// TIA Portal V18 export
FUNCTION_BLOCK "FB10-Condition Check_1"   // FB14, LAD
{ S7_Optimized_Access := 'TRUE' }
VERSION : 0.1
// stored: AutoNumber true, IsIECCheckEnabled false, IsRetainMemResEnabled false, MemoryReserve 100, SetENOAutomatically false, UDAEnableTagReadback false
   VAR_INPUT
      "Time" : DInt;
      "Pump ON delay" : DInt;
      Check_Time { ExternalAccessible := 'False'; ExternalVisible := 'False'; ExternalWritable := 'False'} : DInt;
      Pressure_SP { ExternalAccessible := 'False'; ExternalVisible := 'False'; ExternalWritable := 'False'} : Real;
      Pressure_tolerance { ExternalAccessible := 'False'; ExternalVisible := 'False'; ExternalWritable := 'False'} : Real;
      Current_pressure { ExternalAccessible := 'False'; ExternalVisible := 'False'; ExternalWritable := 'False'} : Real;
      selected { ExternalAccessible := 'False'; ExternalVisible := 'False'; ExternalWritable := 'False'} : Bool;
      "Pressurising Tolerance" : Real;
      Pressurising_SP : Real;
   END_VAR
   VAR_OUTPUT
      "dispensing Time PV" : Int;
      "Checking Time pv" { ExternalAccessible := 'False'; ExternalVisible := 'False'; ExternalWritable := 'False'} : Int;
      Leaktest_ok { ExternalAccessible := 'False'; ExternalVisible := 'False'; ExternalWritable := 'False'} : Bool;
      Leaktest_nok { ExternalAccessible := 'False'; ExternalVisible := 'False'; ExternalWritable := 'False'} : Bool;
      Conditiontest_OK : Bool;
      Conditiontest_NOK { ExternalAccessible := 'False'; ExternalVisible := 'False'; ExternalWritable := 'False'} : Bool;
      "PAT @ installation" : DInt;   // Pressure achieved Time @ Installation
      Test_Data : "Condition_Check";
   END_VAR
   VAR_IN_OUT
      Commissioning_mode : Bool;
      "Start ConditonCheck" : Bool;
      "Stop ConditonCheck" : Bool;
      "ConditonCheck Running" : Bool;
      "ConditonCheck completed" : Bool;
      "ON Gear Pump" : Bool;
      "ON inlet" : Bool;
      Pressurising : Bool;
      run_rev : Bool;
   END_VAR
   VAR
      "dispensing time done" : Bool;
      "dispensing time in sec" : DInt;
      "timer input" : DInt;
      IEC_Timer_0_Instance_1 { S7_SetPoint := 'True'} : TON_TIME;
      IEC_Timer_0_Instance_2 { S7_SetPoint := 'True'} : TON_TIME;
      IEC_Timer_0_Instance_4 { S7_SetPoint := 'True'} : TON_TIME;
      "Press+ve" { ExternalAccessible := 'False'; ExternalVisible := 'False'; ExternalWritable := 'False'; S7_SetPoint := 'True'} : Real;
      "Press-ve" { ExternalAccessible := 'False'; ExternalVisible := 'False'; ExternalWritable := 'False'} : Real;
      IEC_Timer_0_Instance_3 { ExternalAccessible := 'False'; ExternalVisible := 'False'; ExternalWritable := 'False'; S7_SetPoint := 'True'} : TON_TIME;
      Checktime_ms { ExternalAccessible := 'False'; ExternalVisible := 'False'; ExternalWritable := 'False'; S7_SetPoint := 'True'} : DInt;
      Check_timesec { ExternalAccessible := 'False'; ExternalVisible := 'False'; ExternalWritable := 'False'} : DInt;
      temp_ons { ExternalAccessible := 'False'; ExternalVisible := 'False'; ExternalWritable := 'False'} : Bool;
      temp : Array[0..5] of Bool;
      IEC_Timer_0_Instance_5 { S7_SetPoint := 'True'} : TON_TIME;
      "WIth Tolerance" { S7_SetPoint := 'True'} : DInt;
      Pressure_achive_time : DInt;
      Pressure_ok : Bool;
      IEC_Timer_0_Instance { S7_SetPoint := 'True'} : TON_TIME;
      Result { S7_SetPoint := 'True'} : Bool;
      "result temp" : Bool;
      IEC_Timer_0_Instance_6 { S7_SetPoint := 'True'} : TON_TIME;
      Start_cond : Bool;
      IEC_Timer_0_Instance_7 { S7_SetPoint := 'True'} : TON_TIME;
   END_VAR
   VAR_TEMP
      ret : Int;
   END_VAR
   VAR_TEMP   // added for the SCL form of the ladder/FBD networks
      _w1 : Bool;
      _w2 : Bool;
      _w3 : Bool;
      _w4 : Bool;
      _w5 : Bool;
   END_VAR
BEGIN

REGION Network 1
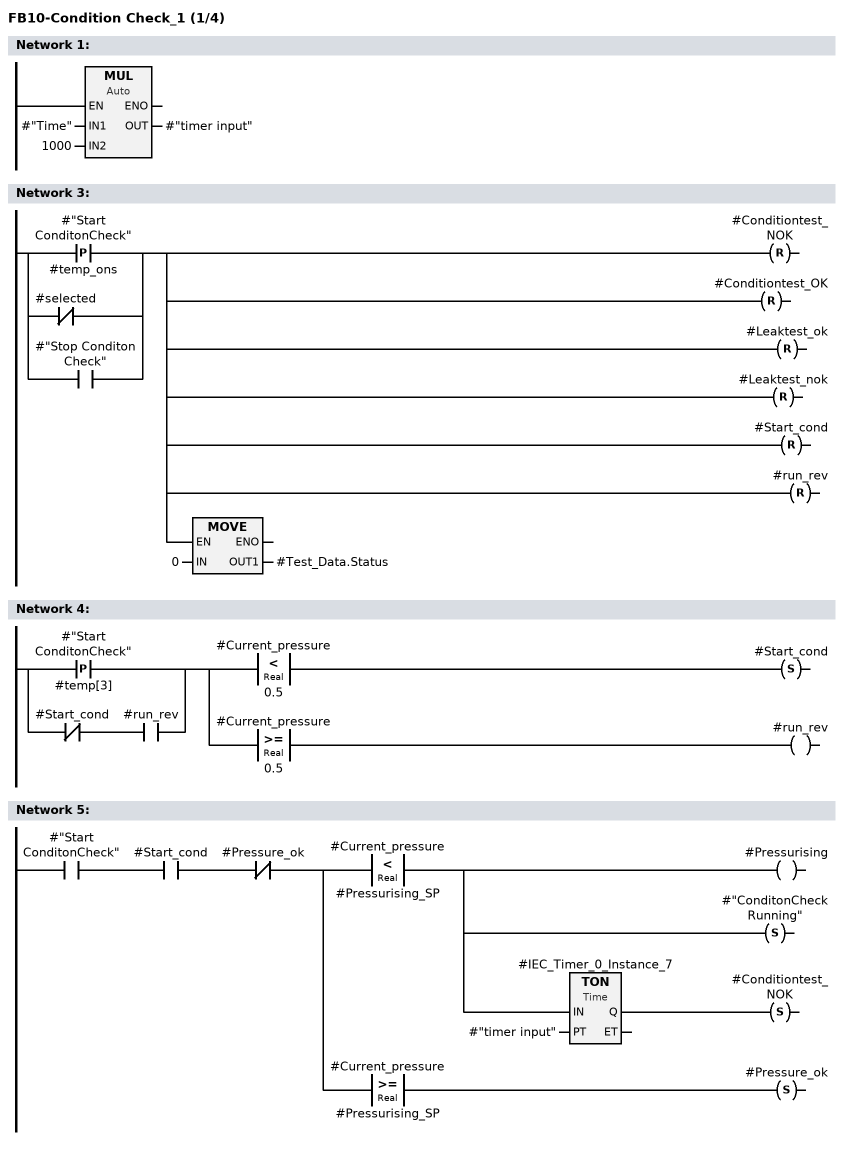
   RUNG wire#powerrail
      Mul(in1 := #"Time", in2 := 1000, out => #"timer input")
   END_RUNG
   // the same network as SCL:
   #"timer input" := #"Time" * 1000;
END_REGION

REGION Network 2 (SCL)
   #"WIth Tolerance" := ROUND(#"PAT @ installation" + ((#"PAT @ installation"*#"Pressurising Tolerance")/100));
END_REGION

REGION Network 3
   RUNG wire#powerrail
      P_Contact(operand := #"Start ConditonCheck", bit := #temp_ons)
      wire#w1
      R_Coil( #Conditiontest_NOK )
   END_RUNG
   RUNG wire#powerrail
      I_Contact( #selected )
   END_RUNG wire#w1
   RUNG wire#powerrail
      Contact( #"Stop ConditonCheck" )
   END_RUNG wire#w1
   RUNG wire#w1
      R_Coil( #Conditiontest_OK )
   END_RUNG
   RUNG wire#w1
      R_Coil( #Leaktest_ok )
   END_RUNG
   RUNG wire#w1
      R_Coil( #Leaktest_nok )
   END_RUNG
   RUNG wire#w1
      R_Coil( #Start_cond )
   END_RUNG
   RUNG wire#w1
      R_Coil( #run_rev )
   END_RUNG
   RUNG wire#w1
      Move(in := 0, out1 => #Test_Data.Status)
   END_RUNG
   // the same network as SCL:
   #_w1 := #"Start ConditonCheck" AND NOT #temp_ons;   // rising edge of #"Start ConditonCheck"
   #temp_ons := #"Start ConditonCheck";
   IF #_w1 OR NOT #selected OR #"Stop ConditonCheck" THEN
       #Conditiontest_NOK := FALSE;
       #Conditiontest_OK := FALSE;
       #Leaktest_ok := FALSE;
       #Leaktest_nok := FALSE;
       #Start_cond := FALSE;
       #run_rev := FALSE;
       #Test_Data.Status := 0;
   END_IF;
END_REGION

REGION Network 4
   RUNG wire#powerrail
      P_Contact(operand := #"Start ConditonCheck", bit := #temp[3])
      wire#w1
      { S7_Templates := "SrcType := Real" } LT_Contact(in1 := #Current_pressure, in2 := 0.5)
      S_Coil( #Start_cond )
   END_RUNG
   RUNG wire#powerrail
      I_Contact( #Start_cond )
      Contact( #run_rev )
   END_RUNG wire#w1
   RUNG wire#w1
      { S7_Templates := "SrcType := Real" } GE_Contact(in1 := #Current_pressure, in2 := 0.5)
      Coil( #run_rev )
   END_RUNG
   // the same network as SCL:
   #_w1 := #"Start ConditonCheck" AND NOT #temp[3];   // rising edge of #"Start ConditonCheck"
   #temp[3] := #"Start ConditonCheck";
   #_w2 := #_w1 OR (NOT #Start_cond AND #run_rev);
   IF #_w2 AND (#Current_pressure < 0.5) THEN #Start_cond := TRUE; END_IF;
   #run_rev := #_w2 AND (#Current_pressure >= 0.5);
END_REGION

REGION Network 5
   RUNG wire#powerrail
      Contact( #"Start ConditonCheck" )
      Contact( #Start_cond )
      I_Contact( #Pressure_ok )
      wire#w1
      { S7_Templates := "SrcType := Real" } LT_Contact(in1 := #Current_pressure, in2 := #Pressurising_SP)
      wire#w2
      Coil( #Pressurising )
   END_RUNG
   RUNG wire#w2
      S_Coil( #"ConditonCheck Running" )
   END_RUNG
   RUNG wire#w2
      { S7_Templates := "time_type := Time" } #IEC_Timer_0_Instance_7.TON(pt := #"timer input", et =>)
      S_Coil( #Conditiontest_NOK )
   END_RUNG
   RUNG wire#w1
      { S7_Templates := "SrcType := Real" } GE_Contact(in1 := #Current_pressure, in2 := #Pressurising_SP)
      S_Coil( #Pressure_ok )
   END_RUNG
   // the same network as SCL:
   #_w1 := #"Start ConditonCheck" AND #Start_cond AND NOT #Pressure_ok;
   #Pressurising := #_w1 AND (#Current_pressure < #Pressurising_SP);
   IF #Pressurising THEN #"ConditonCheck Running" := TRUE; END_IF;
   #IEC_Timer_0_Instance_7(IN := #Pressurising, PT := #"timer input");   // TON
   IF #IEC_Timer_0_Instance_7.Q THEN #Conditiontest_NOK := TRUE; END_IF;
   IF #_w1 AND (#Current_pressure >= #Pressurising_SP) THEN #Pressure_ok := TRUE; END_IF;
END_REGION

REGION Network 6
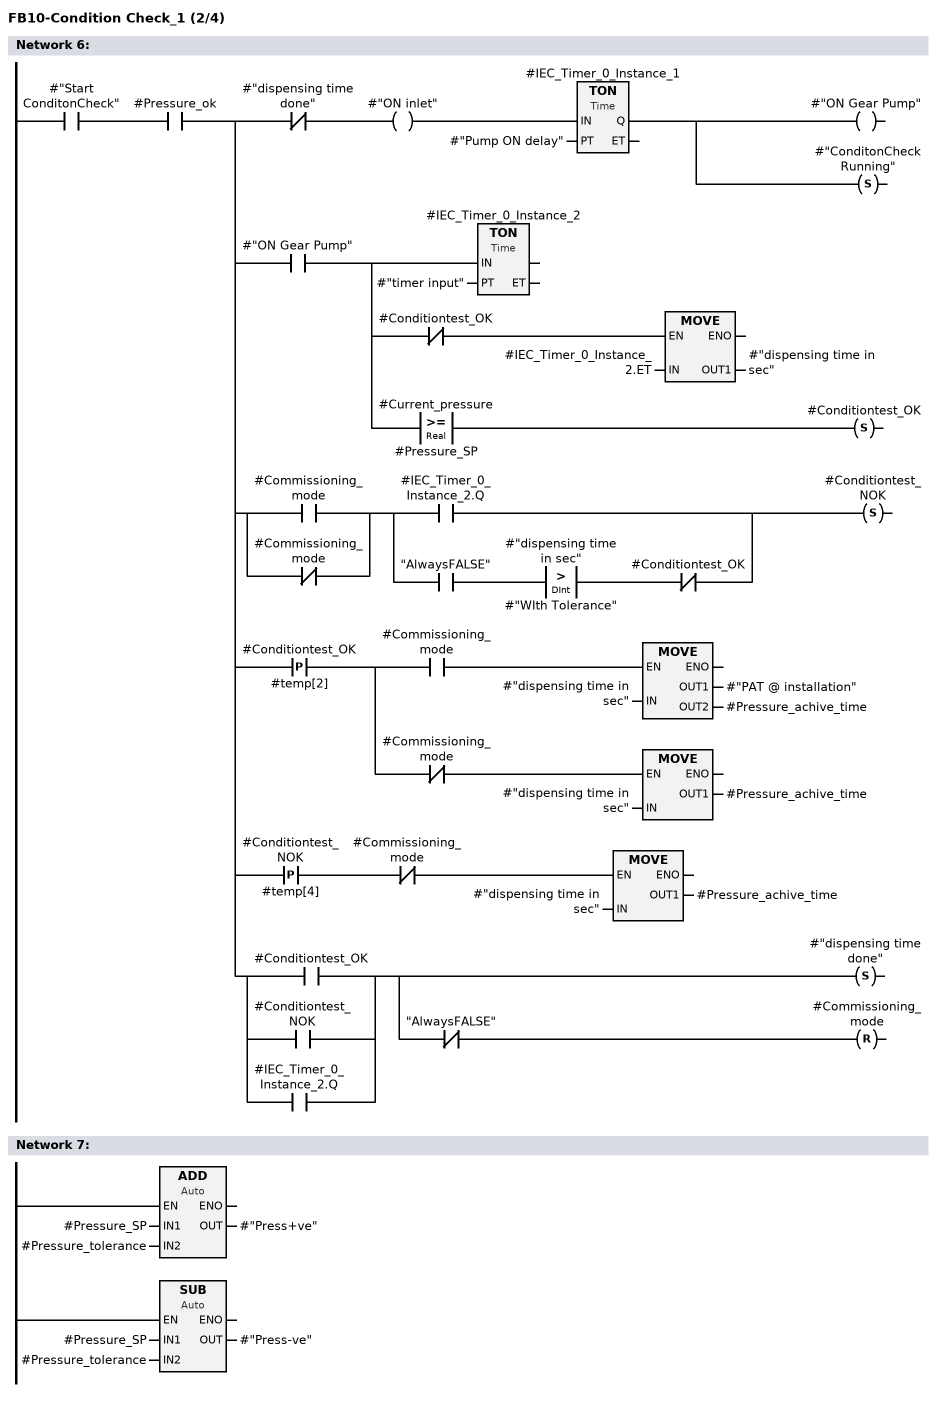
   RUNG wire#powerrail
      Contact( #"Start ConditonCheck" )
      Contact( #Pressure_ok )
      wire#w1
      I_Contact( #"dispensing time done" )
      Coil( #"ON inlet" )
      { S7_Templates := "time_type := Time" } #IEC_Timer_0_Instance_1.TON(pt := #"Pump ON delay", et =>)
      wire#w2
      Coil( #"ON Gear Pump" )
   END_RUNG
   RUNG wire#w2
      S_Coil( #"ConditonCheck Running" )
   END_RUNG
   RUNG wire#w1
      Contact( #"ON Gear Pump" )
      wire#w3
      { S7_Templates := "time_type := Time" } #IEC_Timer_0_Instance_2.TON(pt := #"timer input", et =>)
   END_RUNG
   RUNG wire#w3
      I_Contact( #Conditiontest_OK )
      Move(in := #IEC_Timer_0_Instance_2.ET, out1 => #"dispensing time in sec")
   END_RUNG
   RUNG wire#w3
      { S7_Templates := "SrcType := Real" } GE_Contact(in1 := #Current_pressure, in2 := #Pressure_SP)
      S_Coil( #Conditiontest_OK )
   END_RUNG
   RUNG wire#w1
      Contact( #Commissioning_mode )
      wire#w4
      Contact( #IEC_Timer_0_Instance_2.Q )
      wire#w5
      S_Coil( #Conditiontest_NOK )
   END_RUNG
   RUNG wire#w1
      I_Contact( #Commissioning_mode )
   END_RUNG wire#w4
   RUNG wire#w4
      Contact( "AlwaysFALSE" )
      { S7_Templates := "SrcType := DInt" } GT_Contact(in1 := #"dispensing time in sec", in2 := #"WIth Tolerance")
      I_Contact( #Conditiontest_OK )
   END_RUNG wire#w5
   RUNG wire#w1
      P_Contact(operand := #Conditiontest_OK, bit := #temp[2])
      wire#w6
      Contact( #Commissioning_mode )
      Move(in := #"dispensing time in sec", out1 => #"PAT @ installation", out2 => #Pressure_achive_time)
   END_RUNG
   RUNG wire#w6
      I_Contact( #Commissioning_mode )
      Move(in := #"dispensing time in sec", out1 => #Pressure_achive_time)
   END_RUNG
   RUNG wire#w1
      P_Contact(operand := #Conditiontest_NOK, bit := #temp[4])
      I_Contact( #Commissioning_mode )
      Move(in := #"dispensing time in sec", out1 => #Pressure_achive_time)
   END_RUNG
   RUNG wire#w1
      Contact( #Conditiontest_OK )
      wire#w7
      S_Coil( #"dispensing time done" )
   END_RUNG
   RUNG wire#w1
      Contact( #Conditiontest_NOK )
   END_RUNG wire#w7
   RUNG wire#w1
      Contact( #IEC_Timer_0_Instance_2.Q )
   END_RUNG wire#w7
   RUNG wire#w7
      I_Contact( "AlwaysFALSE" )
      R_Coil( #Commissioning_mode )
   END_RUNG
   // the same network as SCL:
   #_w1 := #"Start ConditonCheck" AND #Pressure_ok;
   #"ON inlet" := #_w1 AND NOT #"dispensing time done";
   #IEC_Timer_0_Instance_1(IN := #"ON inlet", PT := #"Pump ON delay");   // TON
   #"ON Gear Pump" := #IEC_Timer_0_Instance_1.Q;
   IF #IEC_Timer_0_Instance_1.Q THEN #"ConditonCheck Running" := TRUE; END_IF;
   #_w2 := #_w1 AND #"ON Gear Pump";
   #IEC_Timer_0_Instance_2(IN := #_w2, PT := #"timer input");   // TON
   IF #_w2 AND NOT #Conditiontest_OK THEN #"dispensing time in sec" := #IEC_Timer_0_Instance_2.ET; END_IF;
   IF #_w2 AND (#Current_pressure >= #Pressure_SP) THEN #Conditiontest_OK := TRUE; END_IF;
   IF #_w1 AND (#Commissioning_mode OR NOT #Commissioning_mode) AND (#IEC_Timer_0_Instance_2.Q OR ("AlwaysFALSE" AND (#"dispensing time in sec" > #"WIth Tolerance") AND NOT #Conditiontest_OK)) THEN
       #Conditiontest_NOK := TRUE;
   END_IF;
   #_w3 := #_w1 AND #Conditiontest_OK AND NOT #temp[2];   // rising edge of #Conditiontest_OK
   #temp[2] := #Conditiontest_OK;
   IF #_w3 AND #Commissioning_mode THEN
       #"PAT @ installation" := #"dispensing time in sec";
       #Pressure_achive_time := #"dispensing time in sec";
   END_IF;
   IF #_w3 AND NOT #Commissioning_mode THEN #Pressure_achive_time := #"dispensing time in sec"; END_IF;
   #_w4 := #_w1 AND #Conditiontest_NOK AND NOT #temp[4];   // rising edge of #Conditiontest_NOK
   #temp[4] := #Conditiontest_NOK;
   IF #_w4 AND NOT #Commissioning_mode THEN #Pressure_achive_time := #"dispensing time in sec"; END_IF;
   #_w5 := #_w1 AND (#Conditiontest_OK OR #Conditiontest_NOK OR #IEC_Timer_0_Instance_2.Q);
   IF #_w5 THEN #"dispensing time done" := TRUE; END_IF;
   IF #_w5 AND NOT "AlwaysFALSE" THEN #Commissioning_mode := FALSE; END_IF;
END_REGION

REGION Network 7
   RUNG wire#powerrail
      Add(in1 := #Pressure_SP, in2 := #Pressure_tolerance, out => #"Press+ve")
   END_RUNG
   RUNG wire#powerrail
      Sub(in1 := #Pressure_SP, in2 := #Pressure_tolerance, out => #"Press-ve")
   END_RUNG
   // the same network as SCL:
   #"Press+ve" := #Pressure_SP + #Pressure_tolerance;
   #"Press-ve" := #Pressure_SP - #Pressure_tolerance;
END_REGION

REGION Network 8
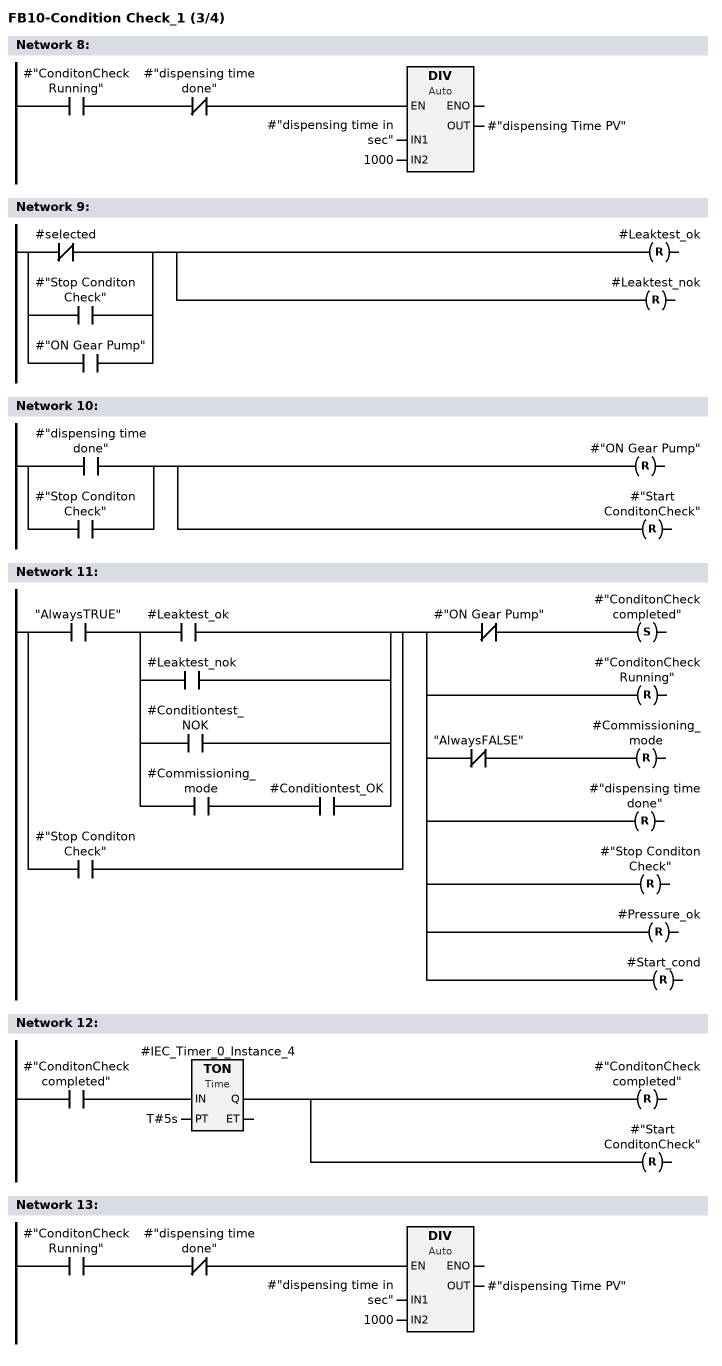
   RUNG wire#powerrail
      Contact( #"ConditonCheck Running" )
      I_Contact( #"dispensing time done" )
      Div(in1 := #"dispensing time in sec", in2 := 1000, out => #"dispensing Time PV")
   END_RUNG
   // the same network as SCL:
   IF #"ConditonCheck Running" AND NOT #"dispensing time done" THEN
       #"dispensing Time PV" := #"dispensing time in sec" / 1000;
   END_IF;
END_REGION

REGION Network 9
   RUNG wire#powerrail
      I_Contact( #selected )
      wire#w1
      R_Coil( #Leaktest_ok )
   END_RUNG
   RUNG wire#powerrail
      Contact( #"Stop ConditonCheck" )
   END_RUNG wire#w1
   RUNG wire#powerrail
      Contact( #"ON Gear Pump" )
   END_RUNG wire#w1
   RUNG wire#w1
      R_Coil( #Leaktest_nok )
   END_RUNG
   // the same network as SCL:
   IF NOT #selected OR #"Stop ConditonCheck" OR #"ON Gear Pump" THEN
       #Leaktest_ok := FALSE;
       #Leaktest_nok := FALSE;
   END_IF;
END_REGION

REGION Network 10
   RUNG wire#powerrail
      Contact( #"dispensing time done" )
      wire#w1
      R_Coil( #"ON Gear Pump" )
   END_RUNG
   RUNG wire#powerrail
      Contact( #"Stop ConditonCheck" )
   END_RUNG wire#w1
   RUNG wire#w1
      R_Coil( #"Start ConditonCheck" )
   END_RUNG
   // the same network as SCL:
   IF #"dispensing time done" OR #"Stop ConditonCheck" THEN
       #"ON Gear Pump" := FALSE;
       #"Start ConditonCheck" := FALSE;
   END_IF;
END_REGION

REGION Network 11
   RUNG wire#powerrail
      Contact( "AlwaysTRUE" )
      wire#w1
      Contact( #Leaktest_ok )
      wire#w2
      I_Contact( #"ON Gear Pump" )
      S_Coil( #"ConditonCheck completed" )
   END_RUNG
   RUNG wire#w1
      Contact( #Leaktest_nok )
   END_RUNG wire#w2
   RUNG wire#w1
      Contact( #Conditiontest_NOK )
   END_RUNG wire#w2
   RUNG wire#w1
      Contact( #Commissioning_mode )
      Contact( #Conditiontest_OK )
   END_RUNG wire#w2
   RUNG wire#powerrail
      Contact( #"Stop ConditonCheck" )
   END_RUNG wire#w2
   RUNG wire#w2
      R_Coil( #"ConditonCheck Running" )
   END_RUNG
   RUNG wire#w2
      I_Contact( "AlwaysFALSE" )
      R_Coil( #Commissioning_mode )
   END_RUNG
   RUNG wire#w2
      R_Coil( #"dispensing time done" )
   END_RUNG
   RUNG wire#w2
      R_Coil( #"Stop ConditonCheck" )
   END_RUNG
   RUNG wire#w2
      R_Coil( #Pressure_ok )
   END_RUNG
   RUNG wire#w2
      R_Coil( #Start_cond )
   END_RUNG
   // the same network as SCL:
   #_w1 := ("AlwaysTRUE" AND (#Leaktest_ok OR #Leaktest_nok OR #Conditiontest_NOK OR (#Commissioning_mode AND #Conditiontest_OK))) OR #"Stop ConditonCheck";
   IF #_w1 AND NOT #"ON Gear Pump" THEN #"ConditonCheck completed" := TRUE; END_IF;
   IF #_w1 THEN #"ConditonCheck Running" := FALSE; END_IF;
   IF #_w1 AND NOT "AlwaysFALSE" THEN #Commissioning_mode := FALSE; END_IF;
   IF #_w1 THEN
       #"dispensing time done" := FALSE;
       #"Stop ConditonCheck" := FALSE;
       #Pressure_ok := FALSE;
       #Start_cond := FALSE;
   END_IF;
END_REGION

REGION Network 12
   RUNG wire#powerrail
      Contact( #"ConditonCheck completed" )
      { S7_Templates := "time_type := Time" } #IEC_Timer_0_Instance_4.TON(pt := T#5s, et =>)
      wire#w1
      R_Coil( #"ConditonCheck completed" )
   END_RUNG
   RUNG wire#w1
      R_Coil( #"Start ConditonCheck" )
   END_RUNG
   // the same network as SCL:
   #IEC_Timer_0_Instance_4(IN := #"ConditonCheck completed", PT := T#5s);   // TON
   IF #IEC_Timer_0_Instance_4.Q THEN
       #"ConditonCheck completed" := FALSE;
       #"Start ConditonCheck" := FALSE;
   END_IF;
END_REGION

REGION Network 13
   RUNG wire#powerrail
      Contact( #"ConditonCheck Running" )
      I_Contact( #"dispensing time done" )
      Div(in1 := #"dispensing time in sec", in2 := 1000, out => #"dispensing Time PV")
   END_RUNG
   // the same network as SCL:
   IF #"ConditonCheck Running" AND NOT #"dispensing time done" THEN
       #"dispensing Time PV" := #"dispensing time in sec" / 1000;
   END_IF;
END_REGION

REGION Network 14
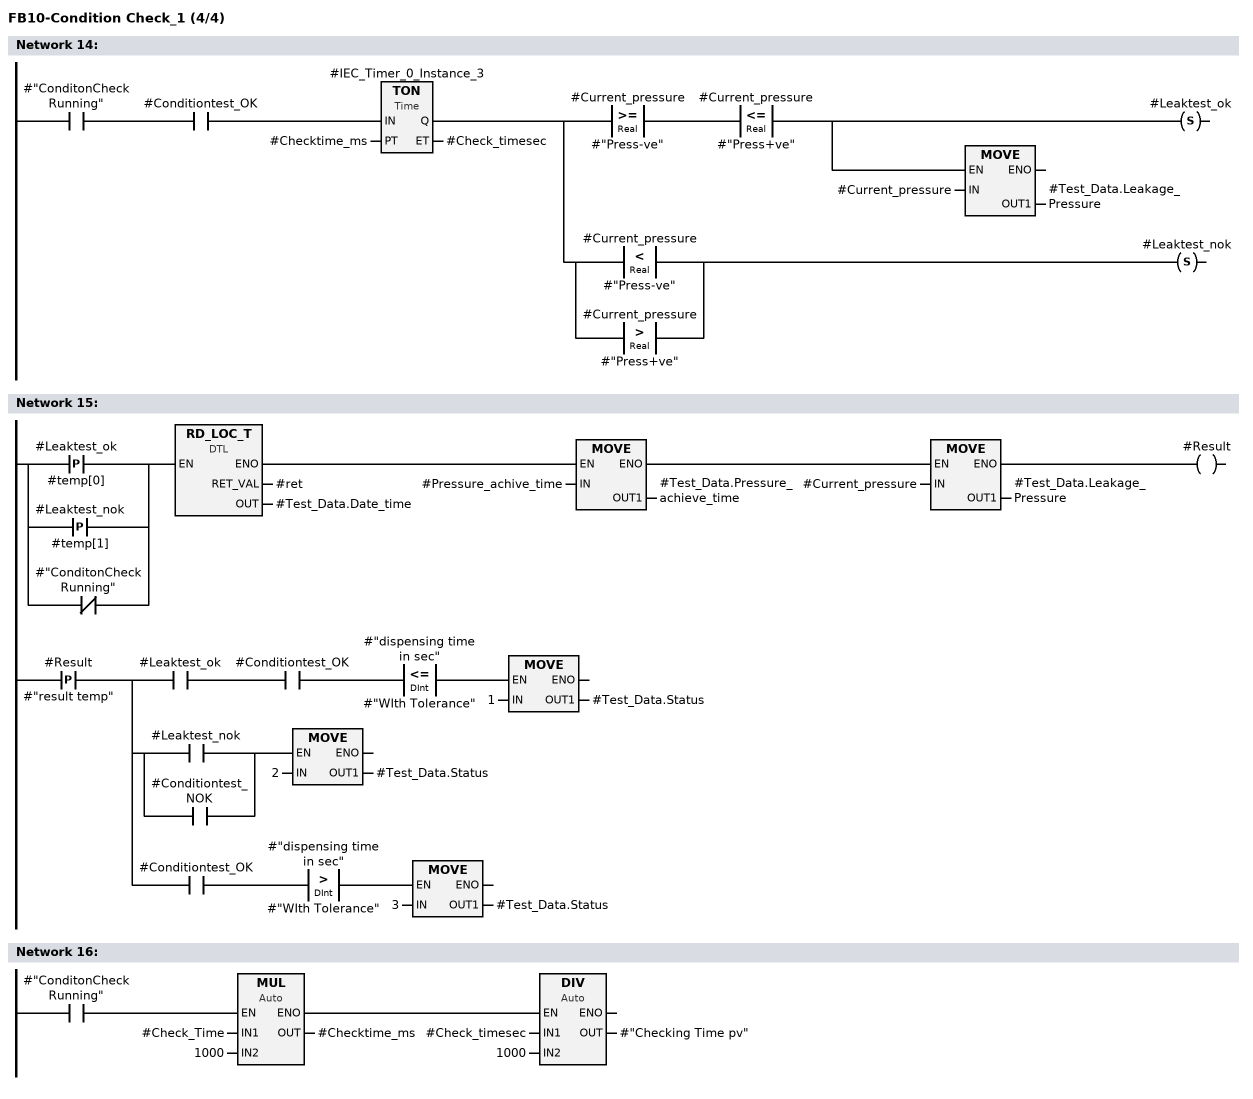
   RUNG wire#powerrail
      Contact( #"ConditonCheck Running" )
      Contact( #Conditiontest_OK )
      { S7_Templates := "time_type := Time" } #IEC_Timer_0_Instance_3.TON(pt := #Checktime_ms, et => #Check_timesec)
      wire#w1
      { S7_Templates := "SrcType := Real" } GE_Contact(in1 := #Current_pressure, in2 := #"Press-ve")
      { S7_Templates := "SrcType := Real" } LE_Contact(in1 := #Current_pressure, in2 := #"Press+ve")
      wire#w2
      S_Coil( #Leaktest_ok )
   END_RUNG
   RUNG wire#w2
      Move(in := #Current_pressure, out1 => #Test_Data.Leakage_Pressure)
   END_RUNG
   RUNG wire#w1
      { S7_Templates := "SrcType := Real" } LT_Contact(in1 := #Current_pressure, in2 := #"Press-ve")
      wire#w3
      S_Coil( #Leaktest_nok )
   END_RUNG
   RUNG wire#w1
      { S7_Templates := "SrcType := Real" } GT_Contact(in1 := #Current_pressure, in2 := #"Press+ve")
   END_RUNG wire#w3
   // the same network as SCL:
   #IEC_Timer_0_Instance_3(IN := #"ConditonCheck Running" AND #Conditiontest_OK,   // TON
                           PT := #Checktime_ms,
                           ET => #Check_timesec);
   IF #IEC_Timer_0_Instance_3.Q AND (#Current_pressure >= #"Press-ve") AND (#Current_pressure <= #"Press+ve") THEN
       #Leaktest_ok := TRUE;
       #Test_Data.Leakage_Pressure := #Current_pressure;
   END_IF;
   IF #IEC_Timer_0_Instance_3.Q AND ((#Current_pressure < #"Press-ve") OR (#Current_pressure > #"Press+ve")) THEN
       #Leaktest_nok := TRUE;
   END_IF;
END_REGION

REGION Network 15
   RUNG wire#powerrail
      P_Contact(operand := #Leaktest_ok, bit := #temp[0])
      wire#w1
      { S7_Templates := "date_type := DTL" } RD_LOC_T(RET_VAL => #ret, OUT => #Test_Data.Date_time)
      Move(in := #Pressure_achive_time, out1 => #Test_Data.Pressure_achieve_time)
      Move(in := #Current_pressure, out1 => #Test_Data.Leakage_Pressure)
      Coil( #Result )
   END_RUNG
   RUNG wire#powerrail
      P_Contact(operand := #Leaktest_nok, bit := #temp[1])
   END_RUNG wire#w1
   RUNG wire#powerrail
      I_Contact( #"ConditonCheck Running" )
   END_RUNG wire#w1
   RUNG wire#powerrail
      P_Contact(operand := #Result, bit := #"result temp")
      wire#w2
      Contact( #Leaktest_ok )
      Contact( #Conditiontest_OK )
      { S7_Templates := "SrcType := DInt" } LE_Contact(in1 := #"dispensing time in sec", in2 := #"WIth Tolerance")
      Move(in := 1, out1 => #Test_Data.Status)
   END_RUNG
   RUNG wire#w2
      Contact( #Leaktest_nok )
      wire#w3
      Move(in := 2, out1 => #Test_Data.Status)
   END_RUNG
   RUNG wire#w2
      Contact( #Conditiontest_NOK )
   END_RUNG wire#w3
   RUNG wire#w2
      Contact( #Conditiontest_OK )
      { S7_Templates := "SrcType := DInt" } GT_Contact(in1 := #"dispensing time in sec", in2 := #"WIth Tolerance")
      Move(in := 3, out1 => #Test_Data.Status)
   END_RUNG
   // the same network as SCL:
   #_w1 := #Leaktest_ok AND NOT #temp[0];   // rising edge of #Leaktest_ok
   #temp[0] := #Leaktest_ok;
   #_w2 := #Leaktest_nok AND NOT #temp[1];   // rising edge of #Leaktest_nok
   #temp[1] := #Leaktest_nok;
   #_w3 := #_w1 OR #_w2 OR NOT #"ConditonCheck Running";
   #ret := RD_LOC_T(EN := #_w3, OUT => #Test_Data.Date_time, ENO => #_w4);
   IF #_w4 THEN
       #Test_Data.Pressure_achieve_time := #Pressure_achive_time;
       #Test_Data.Leakage_Pressure := #Current_pressure;
   END_IF;
   #Result := #_w4;
   #_w5 := #Result AND NOT #"result temp";   // rising edge of #Result
   #"result temp" := #Result;
   IF #_w5 AND #Leaktest_ok AND #Conditiontest_OK AND (#"dispensing time in sec" <= #"WIth Tolerance") THEN
       #Test_Data.Status := 1;
   END_IF;
   IF #_w5 AND (#Leaktest_nok OR #Conditiontest_NOK) THEN #Test_Data.Status := 2; END_IF;
   IF #_w5 AND #Conditiontest_OK AND (#"dispensing time in sec" > #"WIth Tolerance") THEN
       #Test_Data.Status := 3;
   END_IF;
END_REGION

REGION Network 16
   RUNG wire#powerrail
      Contact( #"ConditonCheck Running" )
      Mul(in1 := #Check_Time, in2 := 1000, out => #Checktime_ms)
      Div(in1 := #Check_timesec, in2 := 1000, out => #"Checking Time pv")
   END_RUNG
   // the same network as SCL:
   IF #"ConditonCheck Running" THEN
       #Checktime_ms := #Check_Time * 1000;
       #"Checking Time pv" := #Check_timesec / 1000;
   END_IF;
END_REGION
END_FUNCTION_BLOCK
